// TIA Portal V20 export
// export: Created 2025-12-01T14:56:59.2939452Z, ExportSetting None, DisplayName Totally Integrated Automation Portal, DisplayVersion V20 Update 3, DisplayName TIA Portal Openness, DisplayVersion V20 Update 3, DisplayName TIA Portal Version Control Interface, DisplayVersion V20 Update 3, DisplayName STEP 7 Professional, DisplayVersion V20 Update 3, DisplayName STEP 7 Safety, DisplayVersion V20 Update 2, DisplayName WinCC Basic/Comfort/Advanced, DisplayVersion V20 Update 3, DisplayName WinCC Professional, DisplayVersion V20 Update 3, DisplayName WinCC Unified, DisplayVersion V20 Update 3
FUNCTION "FC401_Conector_Mx_a_TL" : Void   // FC401, LAD
{ S7_Optimized_Access := 'FALSE' }
AUTHOR : TLigero
NAME : 20130323
VERSION : 3.0
// stored: AutoNumber false, SetENOAutomatically false
   VAR_INPUT
      Mesa : UInt;   // Numero de mesa de la funcion de ligero
      AVTF_MAnt_Mx : Bool;   // marca de la función de tracking
      MAnt_Avance : Bool;   // avance del transportador de tracking
      MAnt_DescargaAct : Bool;   // marca de la función de tracking
      PTF_Mx_MSig : Bool;   // marca de la función ligero
      NXT_Avance : Bool;   // avance del transportador ligero
      Rearme_V_Separacion : Bool;
      V_Separacion_T0_1s : UDInt;
   END_VAR
   VAR_OUTPUT
      NXT_AVTF_Conector : Bool;   // aviso para la función de ligero
      NXT_Descarga_Act_conector : Bool;   // descarga para la función de ligero
      PRV_PTF_conector : Bool;   // permiso para la función de tracking
      PRV_FTF_conector : Bool;   // fin para la función de tracking
   END_VAR
   VAR_TEMP
      Separacion_OK : Bool;
   END_VAR
BEGIN

REGION Network 1: contador de separación
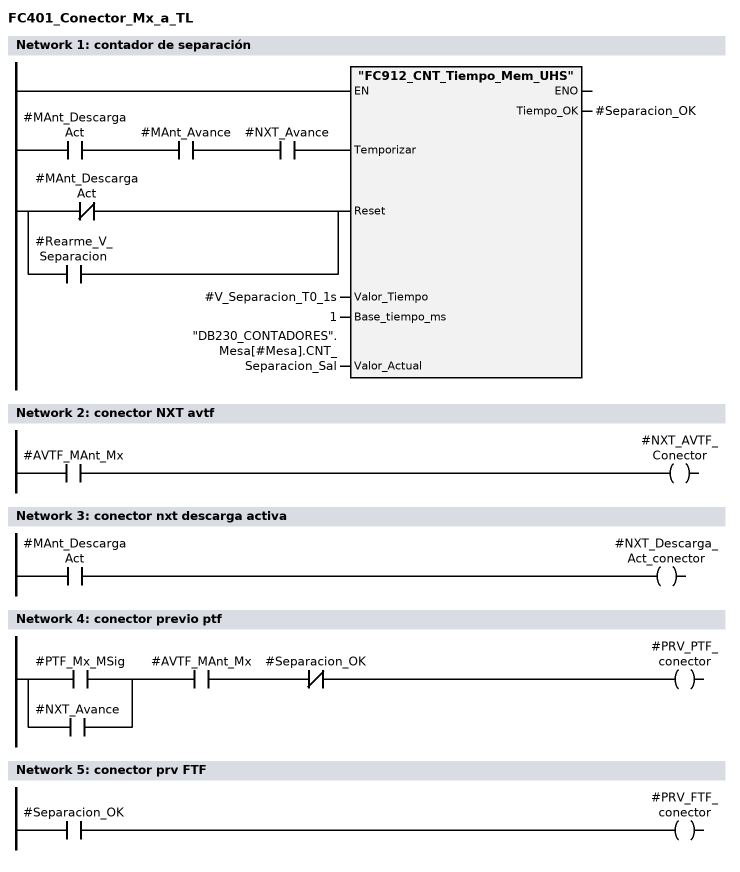
   RUNG wire#powerrail
      "FC912_CNT_Tiempo_Mem_UHS"(Temporizar := wire#w1, Reset := wire#w2, Valor_Tiempo := #V_Separacion_T0_1s, Base_tiempo_ms := 1, Valor_Actual := "DB230_CONTADORES".Mesa[#Mesa].CNT_Separacion_Sal, Tiempo_OK => #Separacion_OK)
   END_RUNG
   RUNG wire#powerrail
      Contact( #MAnt_DescargaAct )
      Contact( #MAnt_Avance )
      Contact( #NXT_Avance )
   END_RUNG wire#w1
   RUNG wire#powerrail
      I_Contact( #MAnt_DescargaAct )
   END_RUNG wire#w2
   RUNG wire#powerrail
      Contact( #Rearme_V_Separacion )
   END_RUNG wire#w2
   // the same network as SCL:
   "FC912_CNT_Tiempo_Mem_UHS"(Temporizar := #MAnt_DescargaAct AND #MAnt_Avance AND #NXT_Avance,
                           Reset := NOT #MAnt_DescargaAct OR #Rearme_V_Separacion,
                           Valor_Tiempo := #V_Separacion_T0_1s,
                           Base_tiempo_ms := 1,
                           Valor_Actual := "DB230_CONTADORES".Mesa[#Mesa].CNT_Separacion_Sal,
                           Tiempo_OK => #Separacion_OK);
END_REGION

REGION Network 2: conector NXT avtf
   RUNG wire#powerrail
      Contact( #AVTF_MAnt_Mx )
      Coil( #NXT_AVTF_Conector )
   END_RUNG
   // the same network as SCL:
   #NXT_AVTF_Conector := #AVTF_MAnt_Mx;
END_REGION

REGION Network 3: conector nxt descarga activa
   RUNG wire#powerrail
      Contact( #MAnt_DescargaAct )
      Coil( #NXT_Descarga_Act_conector )
   END_RUNG
   // the same network as SCL:
   #NXT_Descarga_Act_conector := #MAnt_DescargaAct;
END_REGION

REGION Network 4: conector previo ptf
   RUNG wire#powerrail
      Contact( #PTF_Mx_MSig )
      wire#w1
      Contact( #AVTF_MAnt_Mx )
      I_Contact( #Separacion_OK )
      Coil( #PRV_PTF_conector )
   END_RUNG
   RUNG wire#powerrail
      Contact( #NXT_Avance )
   END_RUNG wire#w1
   // the same network as SCL:
   #PRV_PTF_conector := (#PTF_Mx_MSig OR #NXT_Avance) AND #AVTF_MAnt_Mx AND NOT #Separacion_OK;
END_REGION

REGION Network 5: conector prv FTF
   RUNG wire#powerrail
      Contact( #Separacion_OK )
      Coil( #PRV_FTF_conector )
   END_RUNG
   // the same network as SCL:
   #PRV_FTF_conector := #Separacion_OK;
END_REGION
END_FUNCTION
